(* Tx/Rx (string data) fifo control function block *)
FUNCTION_BLOCK FB_FrameFifo
VAR_INPUT
	bLog: BOOL:= FALSE;(* TRUE => Enable log message output, FALSE => Disable *)
	sPrefix: STRING:= 'Unknown::';(* Log message description string (allows the identification of log message source) *)
	sPut:  STRING;
END_VAR
VAR_OUTPUT
	bOk:BOOL;(* TRUE = New entry added or removed succesfully, FALSE = Fifo overflow or fifo empty *)
	sGet: STRING;
	nCount:UDINT:= 0;(* Number of fifo entries *)
	cbFree:UDINT:= 0;(* Free buffer space *)
	Load:UDINT;
END_VAR
VAR
	fbBuffer 	: FB_MemRingBuffer ;
	buffer		: ARRAY[0..1000] OF STRING;(* Internal buffer memory *)
END_VAR

ACTION AddTail:
(* Adds new fifo entry *)
fbBuffer.A_AddTail( pBuffer:= ADR(buffer), cbBuffer:= SIZEOF(buffer),
					pWrite := ADR( sPut ), cbWrite := SIZEOF( sPut ), 
					bOk=>bOk, nCount=>nCount );
IF bOk THEN
	cbFree := 1000 - fbBuffer.cbSize;(* Calculate the free buffer space *)
	IF bLog THEN(* Log message *)
		ADSLOGSTR( ADSLOG_MSGTYPE_HINT OR ADSLOG_MSGTYPE_LOG, CONCAT( sPrefix, '<="%s"' ),'kk');
	END_IF
END_IF

Load := ((sizeof(buffer) - (sizeof(buffer) -  fbBuffer.cbSize))/sizeof(buffer)) * 100;
END_ACTION

ACTION Clear:
(* Resets fifo = clears all data *)
MEMSET( ADR( sGet ), 0, SIZEOF( sGet ) );
fbBuffer.A_Reset( pBuffer:= ADR(buffer), cbBuffer:= SIZEOF(buffer),
					pWrite := ADR( sPut ), cbWrite := SIZEOF( sPut ), 
					pRead := ADR( sGet ), cbRead := SIZEOF( sGet ),
					bOk=>bOk, nCount=>nCount );
cbFree := 1000;(* Free buffer size *)

Load := sizeof(buffer) - (sizeof(buffer) -  fbBuffer.cbSize) * 100;
END_ACTION

ACTION RemoveHead:
(* Removes oldest fifo entry *)
MEMSET( ADR( sGet ), 0, SIZEOF( sGet ) );
fbBuffer.A_RemoveHead( pBuffer:= ADR(buffer), cbBuffer:= SIZEOF(buffer),
						pRead := ADR( sGet ), cbRead := SIZEOF( sGet ),
						bOk=>bOk, nCount=>nCount );
IF bOk THEN
	cbFree := 1000 - fbBuffer.cbSize;(* Calculate the free buffer space *)
END_IF

Load := sizeof(buffer) - (sizeof(buffer) -  fbBuffer.cbSize) * 100;
END_ACTION

END_FUNCTION_BLOCK

(* stored: Version 1.1.0.1, ProductVersion 3.1.4024.15
   POU FB_FrameFifo: Id {f313e851-f266-44f7-911e-57cc16acbe58}, SpecialFunc None
   Action AddTail: Id {9453fa93-9184-4802-90c5-781861d54553}
   Action Clear: Id {52449281-74cd-4a83-8a85-12ed1bfd2d12}
   Action RemoveHead: Id {bfdcf34c-3cd5-473d-9333-87553dd90971} *)
